FUNCTION_BLOCK CM_SpeedDoor EXTENDS CM_Base IMPLEMENTS I_Door

VAR CONSTANT
	c_MAX_FB_NAME_LENGTH : USINT := 8; //Maximum feedback-name length
END_VAR

VAR_INPUT
	i_stSettings : ST_SettingsSpeedDoor;
	i_bIclkOpen : BOOL := TRUE; //TRUE = interlocked
	i_bIclkClose : BOOL := TRUE; //TRUE = interlocked
	
	i_ref_eCtrlState : REFERENCE TO E_CtrlState;
END_VAR

VAR
	// Inputs
	I_bStaDoorIsOpened AT %I* : BOOL; // Door is opened
	I_bStaDoorIsClosed AT %I* : BOOL; // Door is closed
	I_bStaControllerIsReady AT %I* : BOOL; // Controller is ready (no error)
	
	// Outputs
	Q_bCmdOpen AT %Q* : BOOL; // Command to open door
	Q_bCmdClose AT %Q* : BOOL; // Command to close door
	Q_bCmdReset AT %Q* : BOOL; // Command to reset door (controller)
	
	// Force outputs (IO-test functions)
	s_fbForceCmdReset : FB_ForceOutput;
	s_fbForceCmdOpen : FB_ForceOutput;
	s_fbForceCmdClose : FB_ForceOutput;
	
	// Interlocks
	s_sInterlockedReasonOpen : STRING(GVL.g_MAX_LEN_INTERLOCK_REASON); //External interlocked reason for clarifying reason
	s_sInterlockedReasonClose : STRING(GVL.g_MAX_LEN_INTERLOCK_REASON); //External interlocked reason for clarifying reason
	
	// Interlocks
	s_bIclkOpen : BOOL;
	s_bIclkClose : BOOL;
	
	// Requests
	s_bReqClose : BOOL;
	s_bReqOpen : BOOL;
	s_bReqReset : BOOL;
	
	// Commands
	s_bCmdClose : BOOL;
	s_bCmdOpen : BOOL;
	s_bCmdReset : BOOL;
	
	// States
	s_bStaDoorIsClosed : BOOL;
	s_bStaDoorIsClosing : BOOL;
	s_bStaDoorIsOpened : BOOL;
	s_bStaDoorIsOpening : BOOL;
	s_bStaDoorControllerError : BOOL;
	s_bStaDoorReset : BOOL;
	s_bStaWarning : BOOL;
	
	s_sCfgCloseName : STRING(c_MAX_FB_NAME_LENGTH) := 'Close';
	s_sCfgOpenName : STRING(c_MAX_FB_NAME_LENGTH) := 'Open';
	
	// Alarms	
	s_fbAlarmHandlerDoorController : FB_AlarmHandler;
	s_fbAlarmHandlerOpeningTimeout : FB_AlarmHandler;
	s_fbAlarmHandlerClosingTimeout : FB_AlarmHandler;
	
	s_fbAlarmHandlerOpenInterlocked : FB_AlarmHandler;
	s_fbAlarmHandlerCloseInterlocked : FB_AlarmHandler;
	
	s_errDoorController : BOOL;
	s_errOpeningTimeout : BOOL;
	s_errClosingTimeout : BOOL;
	
	// Timers
	s_tofResetPulse : TOF;
	s_tonOpeningTimeout : TON;
	s_tonClosingTimeout : TON;
	
	//Hmi
	s_stHmiData : ST_SpeedDoor_HMI;
	s_bHmiInit : BOOL := FALSE;
	
	s_fbHmiBtnManualClose : FB_HmiBtn;
	s_fbHmiBtnManualOpen : FB_HmiBtn;
	s_fbHmiBtnManualReset : FB_HmiBtn;
	
	s_fbHmiLedIsClose : FB_HmiLed;
	s_fbHmiLedIsOpen : FB_HmiLed;
	s_fbHmiLedErrorClose : FB_HmiLed;
	s_fbHmiLedErrorOpen : FB_HmiLed;
	s_fbHmiLedErrorController : FB_HmiLed;
	s_fbHmiLedReset : FB_HmiLed;
	
END_VAR


SUPER^();

METHOD PROTECTED _m_Alarms : BOOL

IF NOT SUPER^._m_Alarms() THEN
	RETURN;
END_IF

// Timeout (timers)
s_tonOpeningTimeout(
	IN := i_bReqEnable AND s_bReqOpen AND NOT(s_bStaDoorIsOpened),
	PT := i_stSettings.tDoorOpeningTimeout );
	
s_tonClosingTimeout(
	IN := i_bReqEnable AND s_bReqClose AND NOT(s_bStaDoorIsClosing),
	PT := i_stSettings.tDoorClosingTimeout );
	
// Set error bits
s_errDoorController := i_bReqEnable AND (s_bStaDoorControllerError OR s_errDoorController) AND NOT(i_bCmdReset);
s_errOpeningTimeout := (s_tonOpeningTimeout.Q OR s_errOpeningTimeout) AND NOT(i_bCmdReset);
s_errClosingTimeout := (s_tonClosingTimeout.Q OR s_errClosingTimeout) AND NOT(i_bCmdReset);

// Alarm Handlers
s_fbAlarmHandlerDoorController(
	i_bStaActive := s_errDoorController);
	
s_fbAlarmHandlerOpeningTimeout(
	i_bStaActive := s_errOpeningTimeout);
	
s_fbAlarmHandlerClosingTimeout(
	i_bStaActive := s_errClosingTimeout);
	
// Alarm collector
s_bStaError :=
	s_fbAlarmHandlerDoorController.q_bStaActive
	OR s_fbAlarmHandlerOpeningTimeout.q_bStaActive
	OR s_fbAlarmHandlerClosingTimeout.q_bStaActive;
	
_m_Alarms := TRUE;
END_METHOD

METHOD PROTECTED _m_Devices : BOOL

IF NOT SUPER^._m_Devices() THEN
	RETURN;
END_IF

// Reset request
IF s_bStaDoorIsOpened THEN
	s_bReqOpen := FALSE;
ELSIF s_bStaDoorIsClosed THEN
	s_bReqClose := FALSE;
ELSIF s_bStaError THEN
	s_bReqOpen := FALSE;
	s_bReqClose := FALSE;
END_IF

IF s_fbHmiBtnManualReset.p_osfBtnPress THEN
	s_bReqReset := TRUE;
END_IF

_m_Devices := TRUE;
END_METHOD

METHOD PROTECTED _m_Hmi : BOOL

IF NOT SUPER^._m_Hmi() THEN
	RETURN;
END_IF

//To Hmi
IF NOT(s_bHmiInit) THEN
	//General names
	s_stHmiData.sDescription := i_sCmName;
	
	//Button names
	s_stHmiData.sNameClose := s_fbHmiBtnManualClose.p_sBtnText;
	s_stHmiData.sNameOpen := s_fbHmiBtnManualOpen.p_sBtnText;
	s_stHmiData.sNameReset := s_fbHmiBtnManualReset.p_sBtnText;
	
	s_bHmiInit := TRUE;
END_IF

s_stHmiData.sState := '';

s_stHmiData.bStaOpen := s_bStaDoorIsOpened;
s_stHmiData.bStaClose := s_bStaDoorIsClosed;
s_stHmiData.bStaOpenError := s_fbHmiLedErrorOpen.p_bStaLed;
s_stHmiData.bStaCloseError  := s_fbHmiLedErrorClose.p_bStaLed;
s_stHmiData.bStaError := s_fbHmiLedErrorController.p_bStaLed;
s_stHmiData.bStaReset := s_fbHmiLedReset.p_bStaLed;
s_stHmiData.bBtnOpenEnabled := s_fbHmiBtnManualOpen.p_bStaEnabled;
s_stHmiData.bBtnCloseEnabled := s_fbHmiBtnManualClose.p_bStaEnabled;
s_stHmiData.bBtnResetEnabled := s_fbHmiBtnManualClose.p_bStaEnabled;
s_stHmiData.s_sInterlockedReasonClose := s_sInterlockedReasonClose;
s_stHmiData.s_sInterlockedReasonOpen := s_sInterlockedReasonOpen;

//From Hmi
IF s_stHmiData.bCmdClosePressed THEN
	s_fbHmiBtnManualClose.m_On();
ELSE
	s_fbHmiBtnManualClose.m_Off();
END_IF

IF s_stHmiData.bCmdOpenPressed THEN
	s_fbHmiBtnManualOpen.m_On();
ELSE
	s_fbHmiBtnManualOpen.m_Off();
END_IF

IF s_stHmiData.bCmdResetPressed THEN
	s_fbHmiBtnManualReset.m_On();
ELSE
	s_fbHmiBtnManualReset.m_Off();
END_IF

//Buttons
s_fbHmiBtnManualClose();
s_fbHmiBtnManualOpen();
s_fbHmiBtnManualReset();

//Led
s_fbHmiLedIsClose(i_bStaLed := s_bStaDoorIsClosed);
s_fbHmiLedIsOpen(i_bStaLed := s_bStaDoorIsOpened);
s_fbHmiLedErrorClose(i_bStaLed := s_errClosingTimeout);
s_fbHmiLedErrorOpen(i_bStaLed := s_errOpeningTimeout);
s_fbHmiLedErrorController(i_bStaLed := s_errDoorController);
s_fbHmiLedReset(i_bStaLed := s_bStaDoorReset);

IF __ISVALIDREF(i_ref_eCtrlState) THEN
	//MAINTENANCE-mode is running
	IF (i_eCtrlMode = E_CtrlMode.MAINTENANCE) AND (i_ref_eCtrlState = E_CtrlState.RUNNING) THEN
		s_fbHmiBtnManualClose.p_bStaVisible := TRUE;
		s_fbHmiBtnManualClose.p_bStaEnabled := i_bReqEnable AND NOT(i_bIclkClose);
		
		s_fbHmiBtnManualOpen.p_bStaVisible := TRUE;
		s_fbHmiBtnManualOpen.p_bStaEnabled := i_bReqEnable AND NOT(i_bIclkOpen);
		
		s_fbHmiBtnManualReset.p_bStaVisible := TRUE;
		s_fbHmiBtnManualReset.p_bStaEnabled := i_bReqEnable;
		
		IF s_fbHmiBtnManualClose.p_osrBtnPress THEN
			m_Close();
		END_IF
		
		IF s_fbHmiBtnManualOpen.p_osrBtnPress THEN
			m_Open();
		END_IF
		
		IF s_fbHmiBtnManualReset.p_osrBtnPress THEN
			m_Reset();
		END_IF
		
	//other-mode
	ELSE
		s_fbHmiBtnManualClose.p_bStaVisible := FALSE;
		s_fbHmiBtnManualClose.p_bStaEnabled := FALSE;
		
		s_fbHmiBtnManualOpen.p_bStaVisible := FALSE;
		s_fbHmiBtnManualOpen.p_bStaEnabled := FALSE;
		
		s_fbHmiBtnManualReset.p_bStaVisible := FALSE;
		s_fbHmiBtnManualReset.p_bStaEnabled := FALSE;
	END_IF
END_IF

_m_Hmi := TRUE;
END_METHOD

METHOD PROTECTED _m_Init : BOOL

IF NOT SUPER^._m_Init() THEN
	RETURN;
END_IF

//Alarm config
s_fbAlarmHandlerDoorController.i_eAlarmLevel := E_AlarmLevel.Alarm;
s_fbAlarmHandlerDoorController.i_sAlarmText := CONCAT(i_sCmName , CONCAT(': Controller - ', 'has error (check DYNACO-system).'));

s_fbAlarmHandlerOpeningTimeout.i_eAlarmLevel := E_AlarmLevel.Alarm;
s_fbAlarmHandlerOpeningTimeout.i_sAlarmText := CONCAT(i_sCmName , ': Door - opening timeout (check DYNACO-system).');

s_fbAlarmHandlerClosingTimeout.i_eAlarmLevel := E_AlarmLevel.Alarm;
s_fbAlarmHandlerClosingTimeout.i_sAlarmText := CONCAT(i_sCmName , ': Door - closing timeout (check DYNACO-system).');

{warning '#TODD: Warning below are not used. Delete?'}
s_fbAlarmHandlerCloseInterlocked.i_eAlarmLevel := E_AlarmLevel.Warning;
s_fbAlarmHandlerOpenInterlocked.i_eAlarmLevel := E_AlarmLevel.Warning;

//Hmi
	s_fbHmiBtnManualClose.p_eButtontype := E_HmiButtonType.PUSHBUTTON;
	s_fbHmiBtnManualClose.p_bStaVisible := FALSE;
	s_fbHmiBtnManualClose.p_bStaEnabled := FALSE;
	s_fbHmiBtnManualClose.p_sBtnText := s_sCfgCloseName;
	
	s_fbHmiBtnManualOpen.p_eButtontype := E_HmiButtonType.PUSHBUTTON;
	s_fbHmiBtnManualOpen.p_bStaVisible := FALSE;
	s_fbHmiBtnManualOpen.p_bStaEnabled := FALSE;
	s_fbHmiBtnManualOpen.p_sBtnText := s_sCfgOpenName;
	
	s_fbHmiBtnManualReset.p_eButtontype := E_HmiButtonType.PUSHBUTTON;
	s_fbHmiBtnManualReset.p_bStaVisible := FALSE;
	s_fbHmiBtnManualReset.p_bStaEnabled := FALSE;
	s_fbHmiBtnManualReset.p_sBtnText := 'Reset';
	
	s_fbHmiLedIsClose.p_bStaVisible := FALSE;
	s_fbHmiLedIsClose.p_sToHmiDescriptionLed := CONCAT('Is at: ', s_sCfgCloseName);
	
	s_fbHmiLedIsOpen.p_bStaVisible := FALSE;
	s_fbHmiLedIsOpen.p_sToHmiDescriptionLed := CONCAT('Is at: ', s_sCfgOpenName);
	
	s_fbHmiLedErrorClose.p_bStaVisible := FALSE;
	s_fbHmiLedErrorClose.p_sToHmiDescriptionLed := 'Closing Timeout';
	
	s_fbHmiLedErrorOpen.p_bStaVisible := FALSE;
	s_fbHmiLedErrorOpen.p_sToHmiDescriptionLed := 'Opening Timeout';
	
	s_fbHmiLedErrorController.p_bStaVisible := FALSE;
	s_fbHmiLedErrorController.p_sToHmiDescriptionLed := 'Door Controller Has Error';
	
	s_fbHmiLedReset.p_bStaVisible := FALSE;
	s_fbHmiLedReset.p_sToHmiDescriptionLed := 'Door Controller Reset';
	
_m_Init := TRUE;
END_METHOD

METHOD PROTECTED _m_Inputs : BOOL

IF NOT SUPER^._m_Inputs() THEN
	RETURN;
END_IF

s_bStaDoorIsOpened := I_bStaDoorIsOpened;
s_bStaDoorIsClosed := I_bStaDoorIsClosed;
s_bStaDoorControllerError := NOT(I_bStaControllerIsReady);

s_bIclkOpen := i_bIclkOpen;
s_bIclkClose := i_bIclkClose;

_m_Inputs := TRUE;
END_METHOD

METHOD PROTECTED _m_Outputs : BOOL

IF NOT SUPER^._m_Outputs() THEN
	RETURN;
END_IF

{warning #TODO: Nog bepalen OF het beter is om onderstaande code te verwerken in FB_Force output}
IF __ISVALIDREF(i_ref_eCtrlState) THEN
	IF (i_eCtrlMode <> E_CtrlMode.IO) OR (i_ref_eCtrlState <> E_CtrlState.RUNNING) THEN
		s_fbForceCmdReset.i_eForceValue := E_ForceValue.RELEASED;
		s_fbForceCmdOpen.i_eForceValue := E_ForceValue.RELEASED;
		s_fbForceCmdClose.i_eForceValue := E_ForceValue.RELEASED;
	END_IF
END_IF

// Generate reset pulse for resetting speeddoor controller (via IO)
s_tofResetPulse(
	IN := (i_bCmdReset AND s_bStaDoorControllerError) OR s_bReqReset,
	PT := i_stSettings.tResetPulseDuration);
 	
s_bReqReset := FALSE;

s_bCmdReset := s_tofResetPulse.Q;
s_bCmdOpen := i_bReqEnable AND s_bReqOpen AND NOT(s_bStaDoorIsOpened);
s_bCmdClose := i_bReqEnable AND s_bReqClose AND NOT(s_bStaDoorIsClosed);

s_fbForceCmdReset(
	i_ref_bCmdInput := s_bCmdReset,
	i_ref_bCmdOutput := Q_bCmdReset);
	
s_fbForceCmdOpen(
	i_ref_bCmdInput := s_bCmdOpen,
	i_ref_bCmdOutput := Q_bCmdOpen);
	
s_fbForceCmdClose(
	i_ref_bCmdInput := s_bCmdClose,
	i_ref_bCmdOutput := Q_bCmdClose);
	
s_bStaDoorReset := Q_bCmdReset;
	
_m_Outputs := TRUE;
END_METHOD

METHOD PUBLIC m_Close : BOOL

IF NOT i_bReqEnable THEN
	RETURN;
END_IF

s_bReqClose := TRUE;
s_bReqOpen := FALSE;

m_Close := TRUE;
END_METHOD

METHOD PUBLIC m_Open : BOOL

IF NOT i_bReqEnable THEN
	RETURN;
END_IF

s_bReqClose := FALSE;
s_bReqOpen := TRUE;

m_Open := TRUE;
END_METHOD

METHOD PUBLIC m_Reset : BOOL

IF NOT i_bReqEnable THEN
	RETURN;
END_IF

s_bReqReset := TRUE;

m_Reset := TRUE;
END_METHOD

METHOD PUBLIC m_Stop : BOOL

s_bReqClose := FALSE;
s_bReqOpen := FALSE;

m_Stop := TRUE;
END_METHOD

{attribute 'monitoring':='call'}
PROPERTY PUBLIC p_bStaIsClosed : BOOL
GET

p_bStaIsClosed := s_bStaDoorIsClosed;
END_GET
END_PROPERTY

{attribute 'monitoring':='call'}
PROPERTY PUBLIC p_bStaIsClosing : BOOL
GET

p_bStaIsClosing := s_bReqClose AND NOT(s_bStaDoorIsClosed);
END_GET
END_PROPERTY

{attribute 'monitoring':='call'}
PROPERTY PUBLIC p_bStaIsOpened : BOOL
GET

p_bStaIsOpened := s_bStaDoorIsOpened;
END_GET
END_PROPERTY

{attribute 'monitoring':='call'}
PROPERTY PUBLIC p_bStaIsOpening : BOOL
GET

p_bStaIsOpening := s_bReqOpen AND NOT(s_bStaDoorIsOpened);
END_GET
END_PROPERTY

{attribute 'monitoring':='call'}
PROPERTY PUBLIC p_bStaWarning : BOOL
GET

p_bStaWarning := s_bStaWarning;
END_GET
END_PROPERTY

{attribute 'monitoring':='call'}
PROPERTY PUBLIC p_sCfgCloseName : STRING(c_MAX_FB_NAME_LENGTH)
GET

p_sCfgCloseName := s_sCfgCloseName;
END_GET
SET

s_sCfgCloseName := p_sCfgCloseName;
END_SET
END_PROPERTY

{attribute 'monitoring':='call'}
PROPERTY PUBLIC p_sCfgOpenName : STRING(c_MAX_FB_NAME_LENGTH)
GET

p_sCfgOpenName := s_sCfgOpenName;
END_GET
SET

s_sCfgOpenName := p_sCfgOpenName;
END_SET
END_PROPERTY

{attribute 'monitoring':='call'}
PROPERTY PUBLIC p_sInterlockedReasonClose : STRING(GVL.g_MAX_LEN_INTERLOCK_REASON)
GET

p_sInterlockedReasonClose := s_sInterlockedReasonClose;
END_GET
SET

s_sInterlockedReasonClose := p_sInterlockedReasonClose;
END_SET
END_PROPERTY

{attribute 'monitoring':='call'}
PROPERTY PUBLIC p_sInterlockedReasonOpen : STRING(GVL.g_MAX_LEN_INTERLOCK_REASON)
GET

p_sInterlockedReasonOpen := s_sInterlockedReasonOpen;
END_GET
SET

s_sInterlockedReasonOpen := p_sInterlockedReasonOpen;
END_SET
END_PROPERTY

END_FUNCTION_BLOCK

(* stored: Version 1.1.0.1, ProductVersion 3.1.4024.12
   POU CM_SpeedDoor: Id {e2ac819d-166f-472e-93dd-5b172f53ac70}, SpecialFunc None
   Folder Methods: Id {dd2ef451-5f00-4ad8-b27b-ac26bc262820}
   Folder Base: Id {64eb2fb7-4e3e-4f52-8667-baf2cc40706f}
   Folder Properties: Id {94c06e33-8c98-4e4c-9eed-8612b89d755c}
   Method _m_Alarms: Id {b8083211-2c26-4309-a88e-d066548d2c6f}
   Method _m_Devices: Id {19806151-6bfc-4d1c-84d0-f6d34cd7cf25}
   Method _m_Hmi: Id {7840a539-413d-41f3-9ea8-d8dc0b64e9ee}
   Method _m_Init: Id {ed9edf80-d019-4069-bda1-c3433fdfc559}
   Method _m_Inputs: Id {2072e72c-41a8-4ff9-a497-b847d4491135}
   Method _m_Outputs: Id {b9720cd4-7d4f-42d3-8c4a-83730026236d}
   Method m_Close: Id {7be6b50d-5014-443a-be9d-cc86325ee4dd}
   Method m_Open: Id {49abf2ba-d09f-4bfc-8f29-0007510177f3}
   Method m_Reset: Id {2b94f0b3-4541-4c9a-84a0-3021994a0458}
   Method m_Stop: Id {803f8574-e518-404c-afa9-ff03ca230bc4}
   Property p_bStaIsClosed: Id {ef1dc088-110b-467e-86be-7f52cc54884f}
   Get Get: Id {b33ffe41-405f-44dc-9f2a-e98f9f590f06}
   Property p_bStaIsClosing: Id {e38aff16-9321-443b-af16-44540701eeba}
   Get Get: Id {e9c2334a-530d-42a6-9150-7c6498b38b35}
   Property p_bStaIsOpened: Id {32401d29-e49a-4af3-b091-b0c12d3eebf7}
   Get Get: Id {e6852986-45e6-4621-95cd-f7a435ccbaef}
   Property p_bStaIsOpening: Id {8e8ccc3c-3c29-4ab6-808d-63f7f129183c}
   Get Get: Id {03452541-5f72-4a9e-a064-a4ab86d90405}
   Property p_bStaWarning: Id {21701d96-2825-41a8-848a-46f12da00f82}
   Get Get: Id {be2521da-c152-4c98-b0b3-70c283314d01}
   Property p_sCfgCloseName: Id {80ab1272-73fd-45ad-bf31-7e9fa30658f0}
   Get Get: Id {f0653086-7e22-40cb-8e24-398094960daf}
   Set Set: Id {ac6c8880-1f2b-4819-b18b-1c517b47e40d}
   Property p_sCfgOpenName: Id {b54758bf-ffc1-4a6a-9bf6-cd30b163ccb6}
   Get Get: Id {9822d540-29ce-43e4-a1f6-91fc1bbfa3e8}
   Set Set: Id {93133cab-8c14-4b17-890e-921647c64646}
   Property p_sInterlockedReasonClose: Id {d49da830-0a0f-41b0-b982-a035b2099954}
   Get Get: Id {612fd05c-fec3-4ce9-a783-80fab72135ad}
   Set Set: Id {07feb51c-5a71-418a-b013-80cc34e9028e}
   Property p_sInterlockedReasonOpen: Id {6cfd49fe-dbe4-46e6-bdd6-eb158e1278ff}
   Get Get: Id {1042dd73-2cee-46e7-b3ac-6d91d1034174}
   Set Set: Id {db17fa56-c818-418a-80fd-3222ee07cea2} *)
